TYPE ST_OPC_UANode :
STRUCT
	//struct must be renamed according to convention after deleting old implementation
	NodeID				: ST_UANodeID;
	NodeHdl				: DWORD;
	SizeOfDataType		: UDINT;
	NodeAddInfo			: ST_UANodeAdditionalInfo;
	TargetVar			: POINTER TO BOOL;
END_STRUCT
END_TYPE

(* stored: Version 1.1.0.1, ProductVersion 3.1.4024.10
   DUT ST_OPC_UANode: Id {a0718f54-869e-4ed8-876f-8f6e2e827301} *)
